{attribute 'qualified_only'}
VAR_GLOBAL
	fbTime							: FB_BaseTime;
	fbLocation						: FB_BaseLocation;
	fbLogger						: FB_BaseLogger;
	stCommonData					: ST_BaseCommonData;
	
	(*	Konfiguracja MachineControl	*)
	fbDefaultMachineConfiguration	: FB_MachineDefaultConfiguration;
	fbMachineConfigure				: FB_MCMachineConfigure;
	(*	Element FB_MachineControl - sterowanie stanami i trybami pracy	*)
	fbSaMController					: FB_SaMController;
	(*	Główny element sterujący maszyną - logika pracy					*)
	fbMachineControl				: FB_MCMachineControl;
	
	(*	Konfiguracja HMIManager		*)
	fbDedaultHMIConfiguration		: FB_DefaultHMIConfiguration;
	fbHMIConfigure					: FB_HMIConfigure;
	(*	Główny element sterowania wyświetlaniem na HMI					*)
	fbHMIManager					: FB_HMIManager;
	
	(*	Zmienne zakończenia konfiguracji	*)
	bDefaultInitDone				: BOOL;
	bMachineInitDone				: BOOL;
	
	
END_VAR

(* stored: Version 1.1.0.1
   GVL GVL_SystemVariable: Id {465f00b0-f7bb-09b1-309f-79d544e20801} *)
